FUNCTION_BLOCK ACTUORSbutton
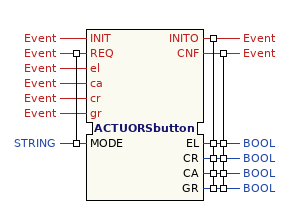
  EVENT_INPUT
    INIT;
    REQ WITH MODE;
    el;
    ca;
    cr;
    gr;
  END_EVENT
  EVENT_OUTPUT
    INITO WITH EL, CA, CR, GR;
    CNF WITH EL, CA, CR, GR;
  END_EVENT
  VAR_INPUT
    MODE : STRING;
  END_VAR
  VAR_OUTPUT
    EL : BOOL;
    CR : BOOL;
    CA : BOOL;
    GR : BOOL;
  END_VAR
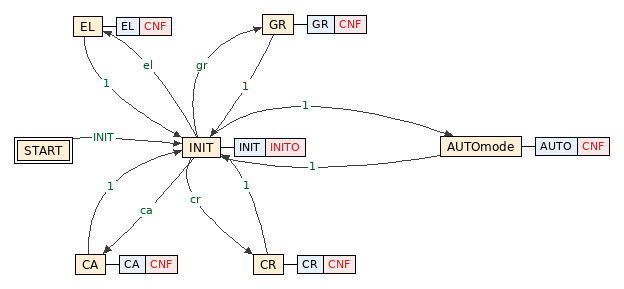
  EC_STATES
    START;
    INIT : INIT -> INITO;
    EL : EL -> CNF;
    CA : CA -> CNF;
    CR : CR -> CNF;
    GR : GR -> CNF;
    AUTOmode : AUTO -> CNF;
  END_STATES
  EC_TRANSITIONS
    START TO INIT := INIT;
    EL TO INIT := 1;
    GR TO INIT := 1;
    CA TO INIT := 1;
    CR TO INIT := 1;
    INIT TO EL := el;
    INIT TO GR := gr;
    INIT TO CA := ca;
    INIT TO CR := cr;
    INIT TO AUTOmode := 1;
    AUTOmode TO INIT := 1;
  END_TRANSITIONS
  ALGORITHM INIT IN ST:
CA := FALSE;&#38;#10;EL := FALSE;&#38;#10;CR := FALSE;&#38;#10;GR := FALSE;&#38;#10;
  END_ALGORITHM
  ALGORITHM EL IN ST:
EL := TRUE;&#38;#10;
  END_ALGORITHM
  ALGORITHM CA IN ST:
CA := TRUE;&#38;#10;
  END_ALGORITHM
  ALGORITHM CR IN ST:
CR := TRUE;&#38;#10;
  END_ALGORITHM
  ALGORITHM GR IN ST:
GR := TRUE;&#38;#10;
  END_ALGORITHM
  ALGORITHM AUTO IN ST:
CA := TRUE;&#38;#10;EL := TRUE;&#38;#10;CR := TRUE;&#38;#10;GR := TRUE;&#38;#10;
  END_ALGORITHM
END_FUNCTION_BLOCK
